FUNCTION_BLOCK FB_BinaryWriter
VAR_INPUT
	i_pDestAddr		: POINTER TO BYTE;
	i_udDestAddrLen	: UDINT;
END_VAR
VAR_OUTPUT
END_VAR
VAR
	pDestAddr		: POINTER TO BYTE;
	udDestAddrLen	: UDINT;
	udCurrentLen 	: UDINT;
END_VAR

METHOD Init : BOOL
VAR_INPUT
	i_pDestAddr		: POINTER TO BYTE;
	i_udDestAddrLen	: UDINT;
END_VAR
pDestAddr 		:= i_pDestAddr;
udDestAddrLen 	:=i_udDestAddrLen;
udCurrentLen 	:= 0;

(* Reset the stream *)
MEMSET(i_pDestAddr, 0, i_udDestAddrLen);
END_METHOD

PROPERTY Length : udint
GET
Length := udCurrentLen;
END_GET
END_PROPERTY

METHOD SetPosition : BOOL
VAR_INPUT
	i_udPosition : UDINT;
END_VAR
IF i_udPosition <= udDestAddrLen THEN
	udCurrentLen := i_udPosition;
	SetPosition := TRUE;
ELSE
	SetPosition := FALSE;
END_IF
END_METHOD

PROPERTY ToString : STRING(255)
GET
VAR
	s255String : STRING(255);
	length : UDINT;
END_VAR
s255String := '';
length := MIN(udCurrentLen, DINT_TO_UDINT(SIZEOF(s255String)));
MEMCPY(ADR(s255String), pDestAddr, length);
ToString := s255String;
END_GET
END_PROPERTY

METHOD WriteString : BOOL
VAR_INPUT
	i_sStringToAppend : T_MaxString;
END_VAR
VAR
	udStringLen: UDINT;
END_VAR

udStringLen := DINT_TO_UDINT(LEN(i_sStringToAppend));

(* Only write if there's memory free for writing *)
IF udCurrentLen + udStringLen < udDestAddrLen THEN
	MEMCPY(pDestAddr + udCurrentLen, ADR(i_sStringToAppend), udStringLen);
	udCurrentLen := udCurrentLen + udStringLen;
	WriteString := TRUE;
ELSE
	WriteString := FALSE;
END_IF
END_METHOD

END_FUNCTION_BLOCK

(* stored: Version 1.1.0.1, ProductVersion 3.1.4020.12
   POU FB_BinaryWriter: Id {05199793-923f-41d0-a5df-80afc16acd51}, SpecialFunc None
   Method Init: Id {7b70c4a0-bc02-45ec-acc9-6aef38d5876d}
   Property Length: Id {d93f15e5-cf65-481e-adfd-9def3caaf26d}
   Get Get: Id {6897a79b-99b8-4674-bc87-2805ff29c529}
   Method SetPosition: Id {375ac408-063a-4dc6-b721-1f8ce21c313f}
   Property ToString: Id {31300ce4-28a7-4508-8ffc-4122ce15a004}
   Get Get: Id {fecd32fc-c098-43dd-b879-42cab6e6e18c}
   Method WriteString: Id {5e836436-21c6-4b75-92df-fe9cac9f7590} *)
